// TIA Portal project "sinior_grad_project" (V18)

(* hardware
DEVICE "S7-1200 station_1"  S7-1200 Station
   slot 0: "Rack_0"  S7-1200 Rack  Rack  V1.0
   slot 1: "PLC_1"  CPU 1214C AC/DC/Rly  6ES7 214-1BG40-0XB0  V4.4
   slot 3: "CB 1241 (RS485)"  CB 1241 (RS485)  6ES7 241-1CH30-1XB0  V1.0
*)

// ===== PLC "PLC_1"  CPU 1214C AC/DC/Rly =====

VAR_GLOBAL   // PLC tag table "Default tag table"
   "PID_PER" AT %MW80 : Int;
   "Ida_Temp" AT %MD10 : Real;
   "Now_temp" AT %MD20 : Real;
   "Now_RPM" AT %MD24 : Real;
   "Port_Err" AT %M28.0 : Bool;
   "Port_Sta" AT %MW32 : Word;
   "USS_Run" AT %M34.0 : Bool;
   "USS_Dri" AT %MW34 : Int;
   "USS_Dir" AT %M36.0 : Bool;
   "RPM_Spd" AT %MD14 : Real;
   "USS_SPD" AT %MD38 : Real;
END_VAR

ORGANIZATION_BLOCK "Cyclic interrupt"   // OB30, LAD, CyclicInterrupt
{ S7_Optimized_Access := 'TRUE' }
VERSION : 0.1
   VAR_INPUT
      Initial_Call : Bool;
      Event_Count : Int;
   END_VAR
BEGIN

REGION Network 1
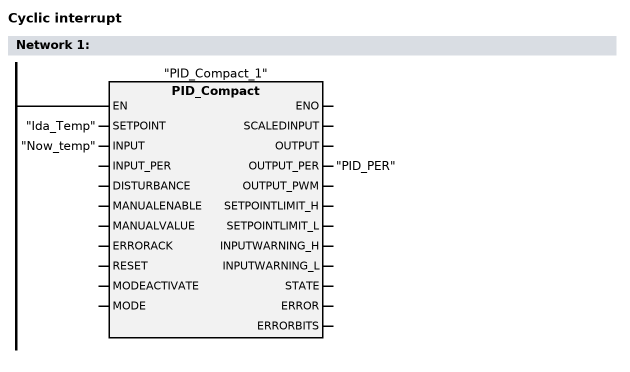
   "PID_Compact_1"(Setpoint := "Ida_Temp", Input := "Now_temp", Output_PER => "PID_PER");   // PID_Compact
END_REGION
END_ORGANIZATION_BLOCK

ORGANIZATION_BLOCK "Cyclic interrupt_1"   // OB31, LAD, CyclicInterrupt
{ S7_Optimized_Access := 'TRUE' }
VERSION : 0.1
   VAR_INPUT
      Initial_Call : Bool;   // Initial call of this OB
      Event_Count : Int;   // Events discarded
   END_VAR
BEGIN

REGION Network 1
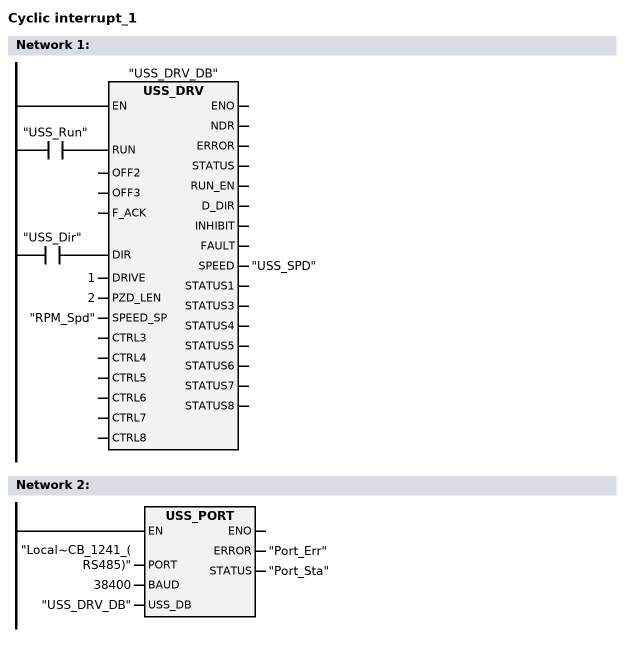
   "USS_DRV_DB"(RUN := "USS_Run",   // USS_DRV
                DIR := "USS_Dir",
                DRIVE := 1,
                PZD_LEN := 2,
                SPEED_SP := "RPM_Spd",
                SPEED => "USS_SPD");
END_REGION

REGION Network 2
   USS_PORT(PORT := "Local~CB_1241_(RS485)",
            BAUD := 38400,
            USS_DB := "USS_DRV_DB",
            ERROR => "Port_Err",
            STATUS => "Port_Sta");
END_REGION
END_ORGANIZATION_BLOCK